FUNCTION_BLOCK FB_Switch EXTENDS FB_LinkDevice
VAR_INPUT		
	nControl  			: BYTE;
END_VAR

VAR_OUTPUT
	nStatus  			: BYTE;
END_VAR

SUPER^();
Control := nControl;
nStatus := Status;

END_FUNCTION_BLOCK

(* stored: Version 1.1.0.1, ProductVersion 3.1.4024.12
   POU FB_Switch: Id {53804fd9-bc27-02f0-3394-255385b99809}, SpecialFunc None *)
